FUNCTION_BLOCK A2X_CLIENT_2_0 (* Send both BOOLs of an A2X adapter as a remote OPC-UA write via CLIENT_2_0, each buffered with an E_D_FF *)
  (* Standard: 61499-2; Description: Copyright (c) 2026 HR Agrartechnik GmbH This program and the accompanying materials are made available under the terms of the Eclipse Public License 2.0 which is available at https://www.eclipse.org/legal/epl-2.0/ SPDX-License-Identifier: EPL-2.0 *)
  (* Version 1.0, 2026-09-05, Franz Höpfinger, HR Agrartechnik GmbH, initial API and implementation and/or initial documentation *)
  PACKAGE adapter::net;
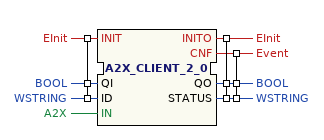
  EVENT_INPUT
    INIT : EInit WITH QI, ID; (* Initialization *)
  END_EVENT
  EVENT_OUTPUT
    INITO : EInit WITH QO, STATUS; (* Initialization Confirm *)
    CNF WITH QO, STATUS; (* Data was sent *)
  END_EVENT
  VAR_INPUT
    QI : BOOL;
    ID : WSTRING;
  END_VAR
  VAR_OUTPUT
    QO : BOOL;
    STATUS : WSTRING;
  END_VAR
  SOCKETS
    IN : adapter::types::unidirectional::A2X; (* UP/DOWN BOOLs to send *)
  END_SOCKETS
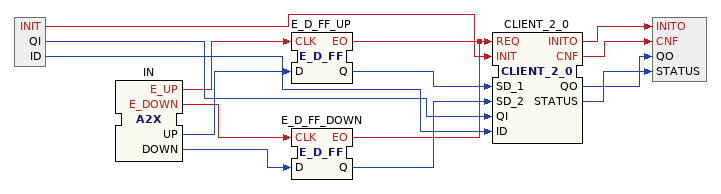
  FBS
    E_D_FF_UP : iec61499::events::E_D_FF;
    E_D_FF_DOWN : iec61499::events::E_D_FF;
    CLIENT_2_0 : iec61499::net::CLIENT_2_0;
  END_FBS
  EVENT_CONNECTIONS
    CLIENT_2_0.INITO TO INITO;
    CLIENT_2_0.CNF TO CNF;
    IN.E_UP TO E_D_FF_UP.CLK;
    IN.E_DOWN TO E_D_FF_DOWN.CLK;
    E_D_FF_UP.EO TO CLIENT_2_0.REQ;
    E_D_FF_DOWN.EO TO CLIENT_2_0.REQ;
    INIT TO CLIENT_2_0.INIT;
  END_CONNECTIONS
  DATA_CONNECTIONS
    CLIENT_2_0.QO TO QO;
    CLIENT_2_0.STATUS TO STATUS;
    IN.UP TO E_D_FF_UP.D;
    IN.DOWN TO E_D_FF_DOWN.D;
    E_D_FF_UP.Q TO CLIENT_2_0.SD_1;
    E_D_FF_DOWN.Q TO CLIENT_2_0.SD_2;
    QI TO CLIENT_2_0.QI;
    ID TO CLIENT_2_0.ID;
  END_CONNECTIONS
END_FUNCTION_BLOCK
